// Mitsubishi GX Works2 project: 0703-공개문제1   PLC: Q02/Q02H

PROGRAM MAIN
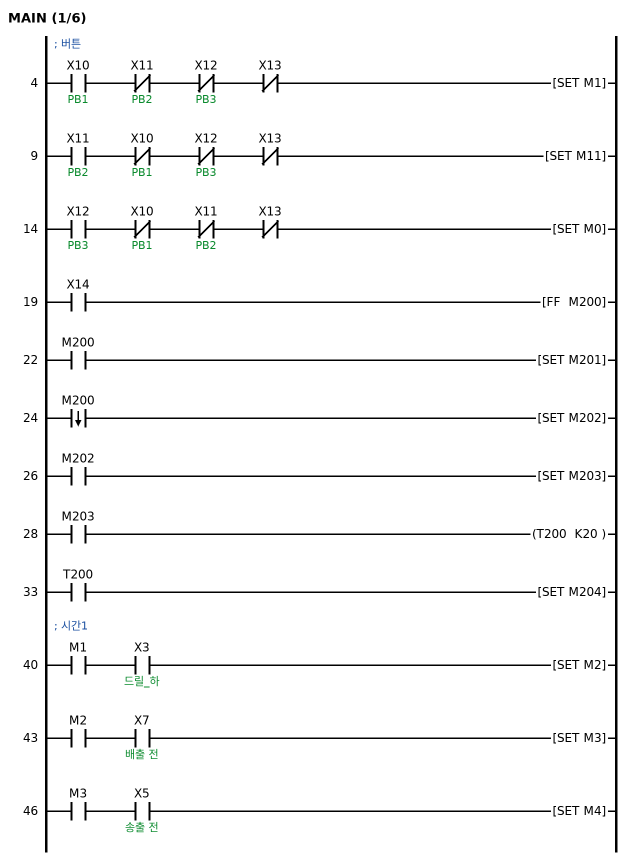
; 버튼
4     LD      X10  ; PB1
      ANI     X11  ; PB2
      ANI     X12  ; PB3
      ANI     X13
      SET     M1
9     LD      X11  ; PB2
      ANI     X10  ; PB1
      ANI     X12  ; PB3
      ANI     X13
      SET     M11
14    LD      X12  ; PB3
      ANI     X10  ; PB1
      ANI     X11  ; PB2
      ANI     X13
      SET     M0
19    LD      X14
      FF      M200
22    LD      M200
      SET     M201
24    LDF     M200
      SET     M202
26    LD      M202
      SET     M203
28    LD      M203
      OUT     T200 K20
33    LD      T200
      SET     M204
; 시간1
40    LD      M1
      AND     X3  ; 드릴_하
      SET     M2
43    LD      M2
      AND     X7  ; 배출 전
      SET     M3
46    LD      M3
      AND     X5  ; 송출 전
      SET     M4
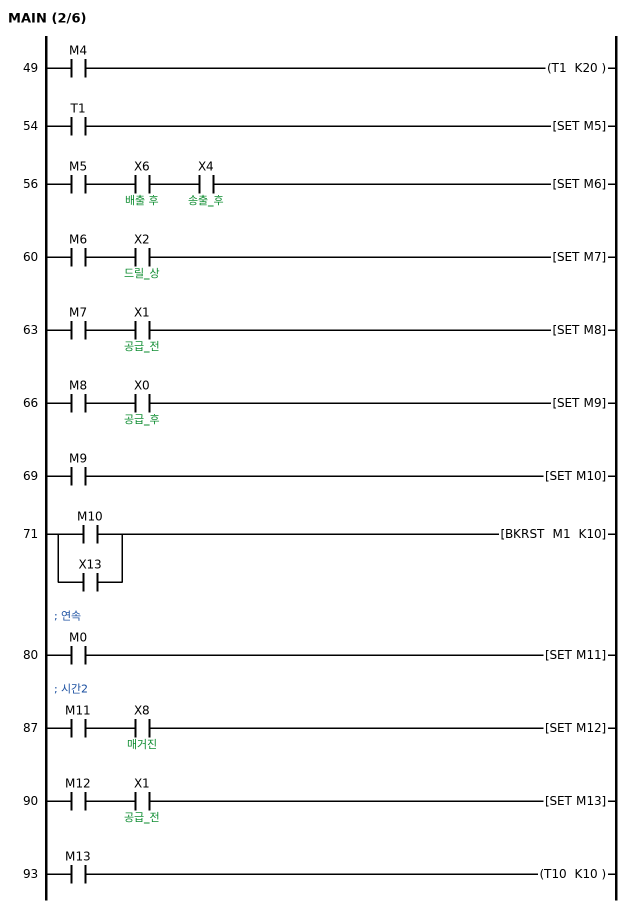
49    LD      M4
      OUT     T1 K20
54    LD      T1
      SET     M5
56    LD      M5
      AND     X6  ; 배출 후
      AND     X4  ; 송출_후
      SET     M6
60    LD      M6
      AND     X2  ; 드릴_상
      SET     M7
63    LD      M7
      AND     X1  ; 공급_전
      SET     M8
66    LD      M8
      AND     X0  ; 공급_후
      SET     M9
69    LD      M9
      SET     M10
71    LD      M10
      OR      X13
      BKRST   M1 K10
; 연속
80    LD      M0
      SET     M11
; 시간2
87    LD      M11
      AND     X8  ; 매거진
      SET     M12
90    LD      M12
      AND     X1  ; 공급_전
      SET     M13
93    LD      M13
      OUT     T10 K10
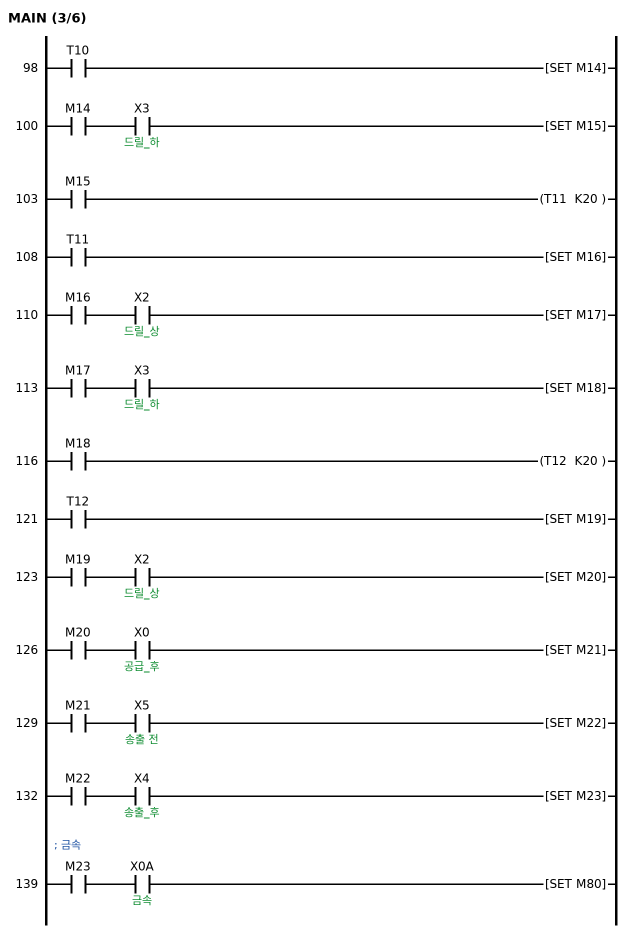
98    LD      T10
      SET     M14
100   LD      M14
      AND     X3  ; 드릴_하
      SET     M15
103   LD      M15
      OUT     T11 K20
108   LD      T11
      SET     M16
110   LD      M16
      AND     X2  ; 드릴_상
      SET     M17
113   LD      M17
      AND     X3  ; 드릴_하
      SET     M18
116   LD      M18
      OUT     T12 K20
121   LD      T12
      SET     M19
123   LD      M19
      AND     X2  ; 드릴_상
      SET     M20
126   LD      M20
      AND     X0  ; 공급_후
      SET     M21
129   LD      M21
      AND     X5  ; 송출 전
      SET     M22
132   LD      M22
      AND     X4  ; 송출_후
      SET     M23
; 금속
139   LD      M23
      AND     X0A  ; 금속
      SET     M80
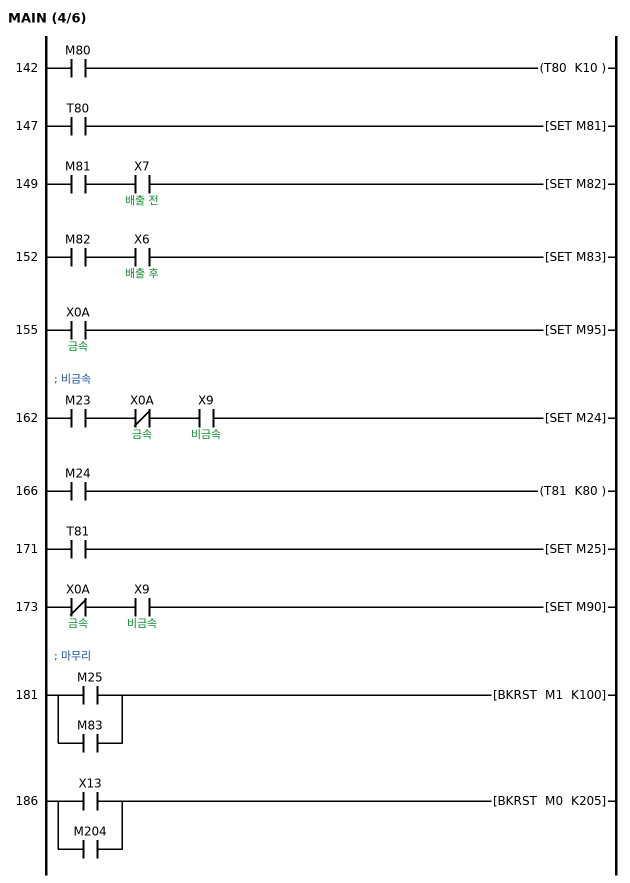
142   LD      M80
      OUT     T80 K10
147   LD      T80
      SET     M81
149   LD      M81
      AND     X7  ; 배출 전
      SET     M82
152   LD      M82
      AND     X6  ; 배출 후
      SET     M83
155   LD      X0A  ; 금속
      SET     M95
; 비금속
162   LD      M23
      ANI     X0A  ; 금속
      AND     X9  ; 비금속
      SET     M24
166   LD      M24
      OUT     T81 K80
171   LD      T81
      SET     M25
173   LDI     X0A  ; 금속
      AND     X9  ; 비금속
      SET     M90
; 마무리
181   LD      M25
      OR      M83
      BKRST   M1 K100
186   LD      X13
      OR      M204
      BKRST   M0 K205
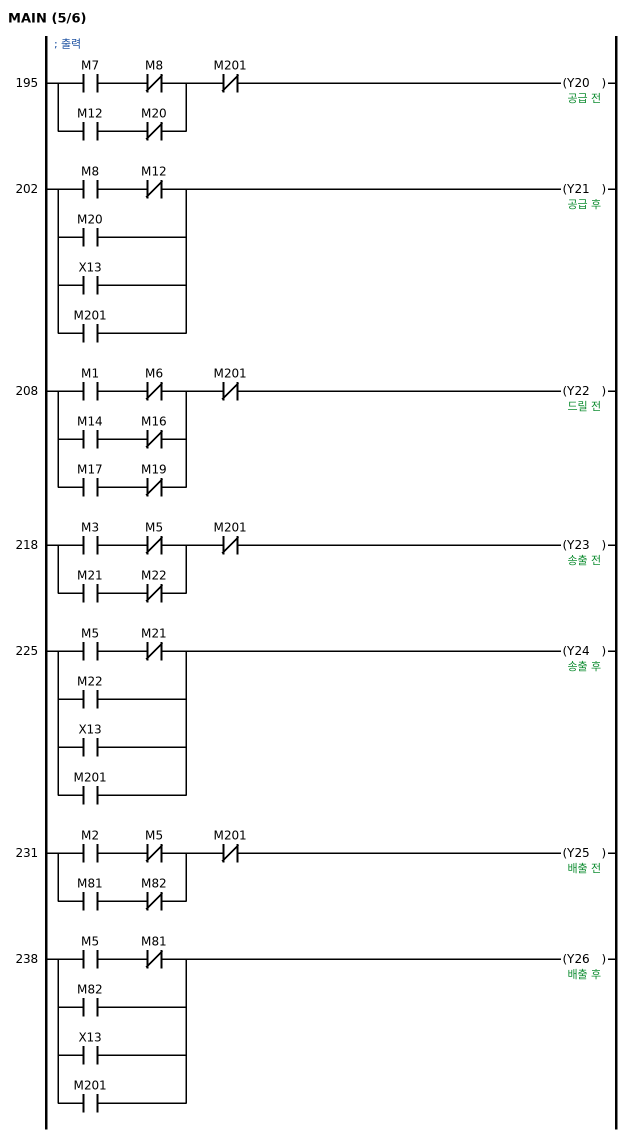
; 출력
195   LD      M7
      ANI     M8
      LD      M12
      ANI     M20
      ORB
      ANI     M201
      OUT     Y20  ; 공급 전
202   LD      M8
      ANI     M12
      OR      M20
      OR      X13
      OR      M201
      OUT     Y21  ; 공급 후
208   LD      M1
      ANI     M6
      LD      M14
      ANI     M16
      ORB
      LD      M17
      ANI     M19
      ORB
      ANI     M201
      OUT     Y22  ; 드릴 전
218   LD      M3
      ANI     M5
      LD      M21
      ANI     M22
      ORB
      ANI     M201
      OUT     Y23  ; 송출 전
225   LD      M5
      ANI     M21
      OR      M22
      OR      X13
      OR      M201
      OUT     Y24  ; 송출 후
231   LD      M2
      ANI     M5
      LD      M81
      ANI     M82
      ORB
      ANI     M201
      OUT     Y25  ; 배출 전
238   LD      M5
      ANI     M81
      OR      M82
      OR      X13
      OR      M201
      OUT     Y26  ; 배출 후
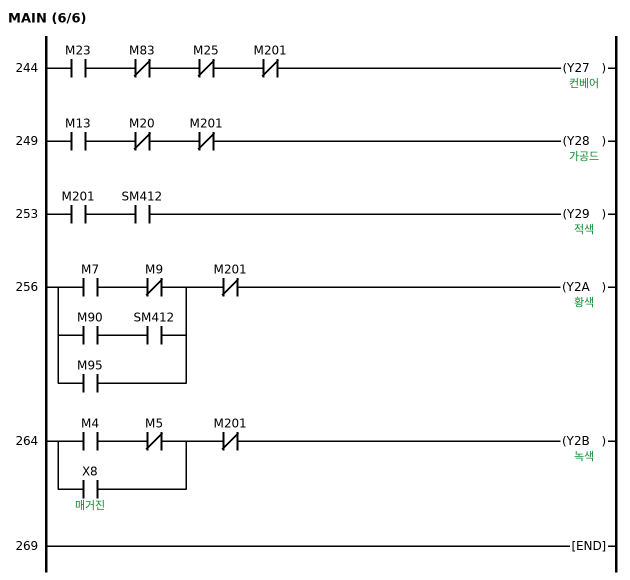
244   LD      M23
      ANI     M83
      ANI     M25
      ANI     M201
      OUT     Y27  ; 컨베어
249   LD      M13
      ANI     M20
      ANI     M201
      OUT     Y28  ; 가공드
253   LD      M201
      AND     SM412
      OUT     Y29  ; 적색
256   LD      M7
      ANI     M9
      LD      M90
      AND     SM412
      ORB
      OR      M95
      ANI     M201
      OUT     Y2A  ; 황색
264   LD      M4
      ANI     M5
      OR      X8  ; 매거진
      ANI     M201
      OUT     Y2B  ; 녹색
269   END
END_PROGRAM

PROGRAM MAIN1
0     END
END_PROGRAM
